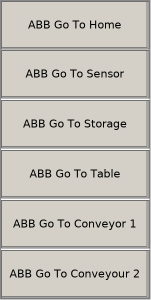
VISUALIZATION _VisuABBGoTo  // 151x300
    Button (1,1 148x48), "ABB Go To Home"
        toggle ComGVL._fbTryOutABBGoToHomeEn
    Button (1,50 148x48), "ABB Go To Sensor"
        toggle ComGVL._fbTryOutABBGoToSensorEn
    Button (1,100 148x48), "ABB Go To Storage"
        toggle ComGVL._fbTryOutABBGoToStorageEn
    Button (1,150 148x48), "ABB Go To Table"
        toggle ComGVL._fbTryOutABBGoToTableEn
    Button (1,200 148x48), "ABB Go To Conveyor 1"
        toggle ComGVL._fbTryOutABBGoToConveyor1En
    Button (1,250 148x48), "ABB Go To Conveyour 2"
        toggle ComGVL._fbTryOutABBGoToConveyor2En
END_VISUALIZATION

(* stored: Version 1.1.0.1, ProductVersion 3.1.4024.2
   Visu _VisuABBGoTo: Id {b776b91d-167b-4588-bc49-9cb3b186e93d} *)
